// TIA Portal V20 export
FUNCTION_BLOCK "Side_Shifter_Auto"   // FB13, LAD
{ S7_Optimized_Access := 'TRUE' }
// stored: MemoryReserve 100, SetENOAutomatically false
   VAR_INPUT
      iSL_Distance : Int;
      iSR_Distance : Int;
      Home_1_SR : Int;
      Home_2_SR : Int;
      Home_1_SL : Int;
      Home_2_SL : Int;
      iGo_H1 : Bool;
      iGo_H2 : Bool;
      ST1_Empty : Bool;
      ST2_Empty : Bool;
      SL_Sen_up : Bool;
      SR_Sen_up : Bool;
   END_VAR
   VAR_OUTPUT
      qSL_Go_Forward : Bool;
      qSL_Go_Backward : Bool;
      qSL_SetSpeed : Int;
      qSR_Go_Forward : Bool;
      qSR_Go_Backward : Bool;
      qSR_SetSpeed : Int;
      qST1_Flash_Sz1 : Bool;
      qST2_Flash_Sz1 : Bool;
      Alarm_Desync : Bool;
      inPosition : Bool;
   END_VAR
   VAR
      targetPosSR : Int;
      targetPosSL : Int;
      moveActive : Bool;
      distanceToTargetSL : Int;
      distanceToTargetSR : Int;
      distanceSL_SR : Int;
      selectedStation : Int;
      maxDelta : Real;
      k_sync : Real;
      deltaClamped : Real;
      Delta : Real;
      moveActive_SL : Bool;
      moveActive_SR : Bool;
      distanceToTarget_SL : Int;
      distanceToTarget_SR : Int;
      NominalOffset : Int;
      syncError : Int;
      baseSpeedSR : Real;
      sensorErrorTimer : TON_TIME;
      pathClear { S7_SetPoint := 'True'} : Bool;
   END_VAR
   VAR_TEMP
      sensorErrorSL : Bool;
      sensorErrorSR : Bool;
      sensorErrorAny : Bool;
      sensorFallback : Bool;
   END_VAR
   VAR CONSTANT
      Tolerance : Int := 3;
      Tolerance_Light : Int := 5;
      Tolerance_Hydro : Int := 15;
      DistanceSlowZone : Int := 600;
      SpeedFast : Int := 1100;
      SpeedSlow : Int := 320;
      K : Real := 1.5;
      MaxOffset : Int := 200;
   END_VAR
BEGIN

REGION Network 1 (SCL)
   // RESET WYJŚĆ

   #qSL_Go_Forward := FALSE;
   #qSL_Go_Backward := FALSE;
   #qSR_Go_Forward := FALSE;
   #qSR_Go_Backward := FALSE;
   #qSL_SetSpeed := 0;
   #qSR_SetSpeed := 0;
   #Alarm_Desync := FALSE;

   // WYBÓR CELU

   IF #iGo_H1 THEN
       #targetPosSL := #Home_1_SL;
       #targetPosSR := #Home_1_SR;
       #moveActive := TRUE;

   ELSIF #iGo_H2 THEN
       #targetPosSL := #Home_2_SL;
       #targetPosSR := #Home_2_SR;
       #moveActive := TRUE;

   ELSE
       #moveActive := FALSE;
   END_IF;

   // SAFETY

   IF NOT "Data_From_Safety".Safety_Active THEN
       #moveActive := FALSE;
   END_IF;

   // RUCH AKTYWNY

   IF #moveActive THEN

       // DETEKCJA BŁĘDU CZUJNIKÓW

       #sensorErrorSL := (#iSL_Distance < 100);
       #sensorErrorSR := (#iSR_Distance < 100);
       #sensorErrorAny := #sensorErrorSL OR #sensorErrorSR;

       #sensorErrorTimer(
                        IN := #sensorErrorAny,
                        PT := T#3s
       );

       // fallback tylko gdy padł JEDEN czujnik
       #sensorFallback :=
       (#sensorErrorSL XOR #sensorErrorSR)
       AND NOT #sensorErrorTimer.Q;


       // DISTANCE (tylko jeśli czujnik OK)

       IF NOT #sensorErrorSL THEN
           #distanceToTargetSL := ABS(#iSL_Distance - #targetPosSL);
       ELSE
           #distanceToTargetSL := 0;
       END_IF;

       IF NOT #sensorErrorSR THEN
           #distanceToTargetSR := ABS(#iSR_Distance - #targetPosSR);
       ELSE
           #distanceToTargetSR := 0;
       END_IF;


       // SL – KIERUNEK I PRĘDKOŚĆ

       IF NOT #sensorErrorSL AND (#distanceToTargetSL > #Tolerance) THEN

           IF #iSL_Distance > #targetPosSL THEN
               #qSL_Go_Forward := TRUE;
           ELSE
               #qSL_Go_Backward := TRUE;
           END_IF;

           IF #distanceToTargetSL <= #DistanceSlowZone THEN
               #qSL_SetSpeed := #SpeedSlow;
           ELSE
               #qSL_SetSpeed := #SpeedFast;
           END_IF;
       ELSE

           // DOJECHAŁ
           #qSL_SetSpeed := 0;
           #qSL_Go_Forward := FALSE;
           #qSL_Go_Backward := FALSE;
       END_IF;



       // SR – KIERUNEK I PRĘDKOŚĆ BAZOWA

       IF NOT #sensorErrorSR AND (#distanceToTargetSR > #Tolerance) THEN

           IF #iSR_Distance > #targetPosSR THEN
               #qSR_Go_Forward := TRUE;
           ELSE
               #qSR_Go_Backward := TRUE;
           END_IF;

           IF #distanceToTargetSR <= #DistanceSlowZone THEN
               #baseSpeedSR := #SpeedSlow;
           ELSE
               #baseSpeedSR := #SpeedFast;
           END_IF;
           #qSR_SetSpeed := #baseSpeedSR;;

       ELSE
           #qSR_SetSpeed := 0;
           #qSR_Go_Forward := FALSE;
           #qSR_Go_Backward := FALSE;
       END_IF;

       // SPRAWDZ KOLIZJE PRZY PRZEJEZDZIE DLA SL

       #pathClear := TRUE;

       IF #qSL_Go_Forward THEN

           IF ((#Home_1_SL < (#iSL_Distance - #Tolerance_Hydro)) AND (#Home_1_SL > #targetPosSL) AND NOT #ST1_Empty)
               OR ((#Home_2_SL < (#iSL_Distance - #Tolerance_Hydro)) AND (#Home_2_SL > #targetPosSL) AND NOT #ST2_Empty) THEN

               #pathClear := FALSE;

           END_IF;

       END_IF;



       IF #qSL_Go_Backward THEN

           IF ((#Home_1_SL > (#iSL_Distance + #Tolerance_Hydro)) AND (#Home_1_SL < #targetPosSL) AND NOT #ST1_Empty)
               OR ((#Home_2_SL > (#iSL_Distance + #Tolerance_Hydro)) AND (#Home_2_SL < #targetPosSL) AND NOT #ST2_Empty) THEN

               #pathClear := FALSE;

           END_IF;

       END_IF;

       // SYNCHRONIZACJA (TYLKO BEZ FALLBACKU)

       IF NOT #sensorFallback AND (#distanceToTargetSL > #Tolerance) AND (#distanceToTargetSR > #Tolerance) THEN

           #NominalOffset := #targetPosSR - #targetPosSL;
           #syncError := (#iSR_Distance - #iSL_Distance) - #NominalOffset;

           IF ABS(#syncError) > #MaxOffset THEN
               #qSL_Go_Forward := FALSE;
               #qSL_Go_Backward := FALSE;
               #qSR_Go_Forward := FALSE;
               #qSR_Go_Backward := FALSE;
               #qSL_SetSpeed := 0;
               #qSR_SetSpeed := 0;
               #Alarm_Desync := TRUE;
               #moveActive := FALSE;
           END_IF;

           #Delta := #syncError * #k_sync;

           IF #Delta > 300 THEN
               #Delta := 300;
           ELSIF #Delta < -300 THEN
               #Delta := -300;
           END_IF;

           #qSR_SetSpeed := #baseSpeedSR - #Delta;

           IF #qSR_SetSpeed > 1500 THEN
               #qSR_SetSpeed := 1500;
           ELSIF #qSR_SetSpeed < 200 AND #qSR_SetSpeed > 0 THEN
               #qSR_SetSpeed := 200;
           END_IF;

       END_IF;

       // FALLBACK – DWUKIERUNKOWY

       IF #sensorFallback THEN

           // SR padł → SR kopiuje SL
           IF #sensorErrorSR THEN
               #qSR_SetSpeed := #qSL_SetSpeed;
               #qSR_Go_Forward := #qSL_Go_Forward;
               #qSR_Go_Backward := #qSL_Go_Backward;
           END_IF;

           // SL padł → SL kopiuje SR
           IF #sensorErrorSL THEN
               #qSL_SetSpeed := #qSR_SetSpeed;
               #qSL_Go_Forward := #qSR_Go_Forward;
               #qSL_Go_Backward := #qSR_Go_Backward;
           END_IF;

       END_IF;

       // STOP JEŚLI BŁĄD > time

       IF #sensorErrorTimer.Q THEN
           #qSL_Go_Forward := FALSE;
           #qSL_Go_Backward := FALSE;
           #qSR_Go_Forward := FALSE;
           #qSR_Go_Backward := FALSE;
           #qSL_SetSpeed := 0;
           #qSR_SetSpeed := 0;
           #Alarm_Desync := TRUE;
           #moveActive := FALSE;
       END_IF;

       // ZAKOŃCZENIE RUCHU

       IF (NOT #sensorErrorSL) AND (NOT #sensorErrorSR) THEN
           IF (#distanceToTargetSL <= #Tolerance)
               AND (#distanceToTargetSR <= #Tolerance) THEN
               #moveActive := FALSE;
           END_IF;
       END_IF;

   END_IF;

   //BLOKUJ RUCH JESLI KOLIZJA
   IF NOT #pathClear AND #SR_Sen_up AND #SL_Sen_up THEN

       #qSL_Go_Forward := FALSE;
       #qSL_Go_Backward := FALSE;
       #qSR_Go_Forward := FALSE;
       #qSR_Go_Backward := FALSE;

       #qSL_SetSpeed := 0;
       #qSR_SetSpeed := 0;

       #moveActive := FALSE;

   END_IF;


   // IN POSITION

   #inPosition :=
   (NOT #sensorErrorSL) AND (NOT #sensorErrorSR)
   AND (ABS(#iSL_Distance - #targetPosSL) <= #Tolerance_Hydro)
   AND (ABS(#iSR_Distance - #targetPosSR) <= #Tolerance_Hydro);

   // MIGANIE LAMPEK – PRZYCISK TRZYMANY + RUCH

   IF #moveActive AND "Clock_2Hz" THEN

       #qST1_Flash_Sz1 := #iGo_H1;

       #qST2_Flash_Sz1 := #iGo_H2;

   ELSE
       #qST1_Flash_Sz1 := 0;
       #qST2_Flash_Sz1 := 0;

   END_IF;

   // LAMPKI – DOJECHANO DO POZYCJI

   IF #inPosition THEN
       IF ABS(#iSL_Distance - #Home_1_SL) <= #Tolerance_Light
           AND ABS(#iSR_Distance - #Home_1_SR) <= #Tolerance_Light THEN
           #qST1_Flash_Sz1 := 1;

       ELSIF ABS(#iSL_Distance - #Home_2_SL) <= #Tolerance_Light
           AND ABS(#iSR_Distance - #Home_2_SR) <= #Tolerance_Light THEN
           #qST2_Flash_Sz1 := 1;

       END_IF;
   END_IF;
END_REGION
END_FUNCTION_BLOCK
